// TIA Portal V15.1 export
// export: Created 2024-05-17T05:38:24.0424637Z, ExportSetting WithDefaults, DisplayName Totally Integrated Automation Portal, DisplayVersion V15.1 Update 5, DisplayName TIA Portal Openness, DisplayVersion V15.1 Update 5, DisplayName SINAMICS Startdrive Advanced, DisplayVersion V15.1, DisplayName G130, G150, S120, S150, SINAMICS MV, S210, DisplayVersion V15.1, DisplayName G110M, G120, G120C, G120D, G120P, DisplayVersion V15.1, DisplayName STEP 7 Professional, DisplayVersion V15.1 Update 5, DisplayName STEP 7 Safety, DisplayVersion V15.1, DisplayName WinCC Professional, DisplayVersion V15.1 Update 5, DisplayName SIMATIC Visualization Architect, DisplayVersion V15.1
FUNCTION "F209220ZS01Output" : Void   // FC7022, F_FBD
TITLE = Safety Inputs ZMProc / Safety Outputs 209220ZS01
{ S7_Optimized_Access := 'TRUE' }
VERSION : 0.1
// stored: AutoNumber false, IsIECCheckEnabled false, UDAEnableTagReadback false
BEGIN

REGION Network 1: **** --------------------- Infeed Roller // 220CR21 --------------------- ****
END_REGION

REGION Network 2: **** 8 - Outputs **** 209000AK04M1-UE140 Power OFF - 220CR21M1
   // SEW Drive Power OFF
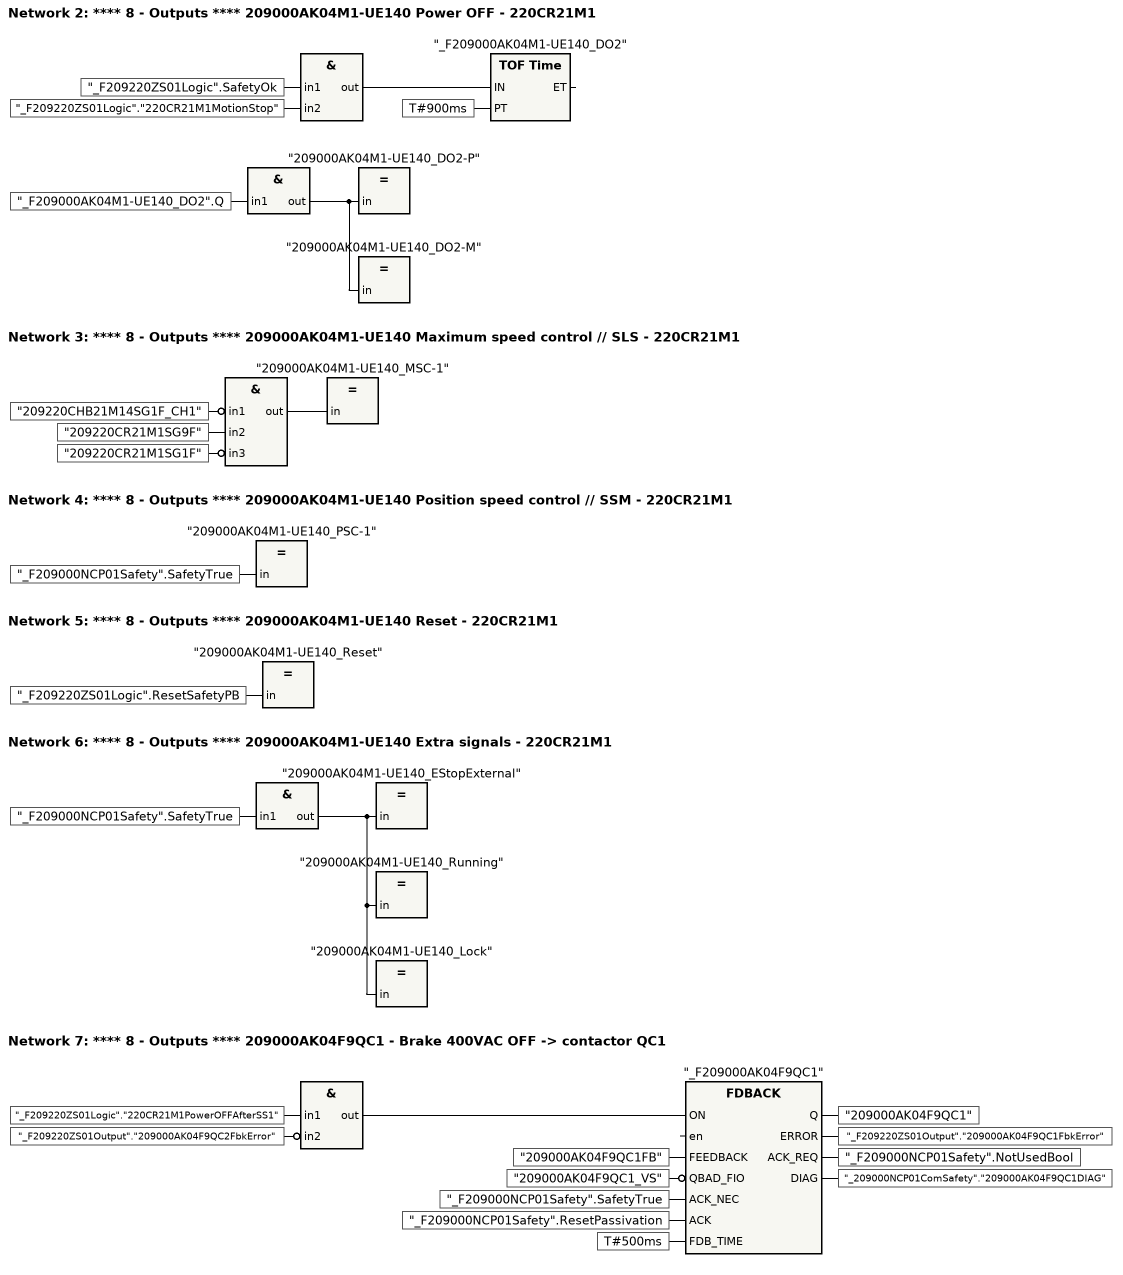
   "_F209000AK04M1-UE140_DO2".TOF(IN := "_F209220ZS01Logic".SafetyOk AND "_F209220ZS01Logic"."220CR21M1MotionStop",
                           PT := T#900ms);
   "209000AK04M1-UE140_DO2-P" := "_F209000AK04M1-UE140_DO2".Q;
   "209000AK04M1-UE140_DO2-M" := "_F209000AK04M1-UE140_DO2".Q;
END_REGION

REGION Network 3: **** 8 - Outputs **** 209000AK04M1-UE140 Maximum speed control // SLS - 220CR21M1
   // SEW Drive Maximum speed control
   "209000AK04M1-UE140_MSC-1" := NOT "209220CHB21M14SG1F_CH1" AND "209220CR21M1SG9F" AND NOT "209220CR21M1SG1F";
END_REGION

REGION Network 4: **** 8 - Outputs **** 209000AK04M1-UE140 Position speed control // SSM - 220CR21M1
   "209000AK04M1-UE140_PSC-1" := "_F209000NCP01Safety".SafetyTrue;
END_REGION

REGION Network 5: **** 8 - Outputs **** 209000AK04M1-UE140 Reset - 220CR21M1
   // SEW Drive Reset
   "209000AK04M1-UE140_Reset" := "_F209220ZS01Logic".ResetSafetyPB;
END_REGION

REGION Network 6: **** 8 - Outputs **** 209000AK04M1-UE140 Extra signals - 220CR21M1
   // SEW Drive Extra signals
   "209000AK04M1-UE140_EStopExternal" := "_F209000NCP01Safety".SafetyTrue;
   "209000AK04M1-UE140_Running" := "_F209000NCP01Safety".SafetyTrue;
   "209000AK04M1-UE140_Lock" := "_F209000NCP01Safety".SafetyTrue;
END_REGION

REGION Network 7: **** 8 - Outputs **** 209000AK04F9QC1 - Brake 400VAC OFF -> contactor QC1
   // Brake 400VAC OFF
   "_F209000AK04F9QC1"(ON := "_F209220ZS01Logic"."220CR21M1PowerOFFAfterSS1" AND NOT "_F209220ZS01Output"."209000AK04F9QC2FbkError",   // FDBACK
                       FEEDBACK := "209000AK04F9QC1FB",
                       QBAD_FIO := NOT "209000AK04F9QC1_VS",
                       ACK_NEC := "_F209000NCP01Safety".SafetyTrue,
                       ACK := "_F209000NCP01Safety".ResetPassivation,
                       FDB_TIME := T#500ms,
                       Q => "209000AK04F9QC1",
                       ERROR => "_F209220ZS01Output"."209000AK04F9QC1FbkError",
                       ACK_REQ => "_F209000NCP01Safety".NotUsedBool,
                       DIAG => "_209000NCP01ComSafety"."209000AK04F9QC1DIAG");
END_REGION

REGION Network 8: **** 8 - Outputs **** 209000AK04F9QC2 - Brake 400VAC OFF -> contactor QC2
   // Brake 400VAC OFF
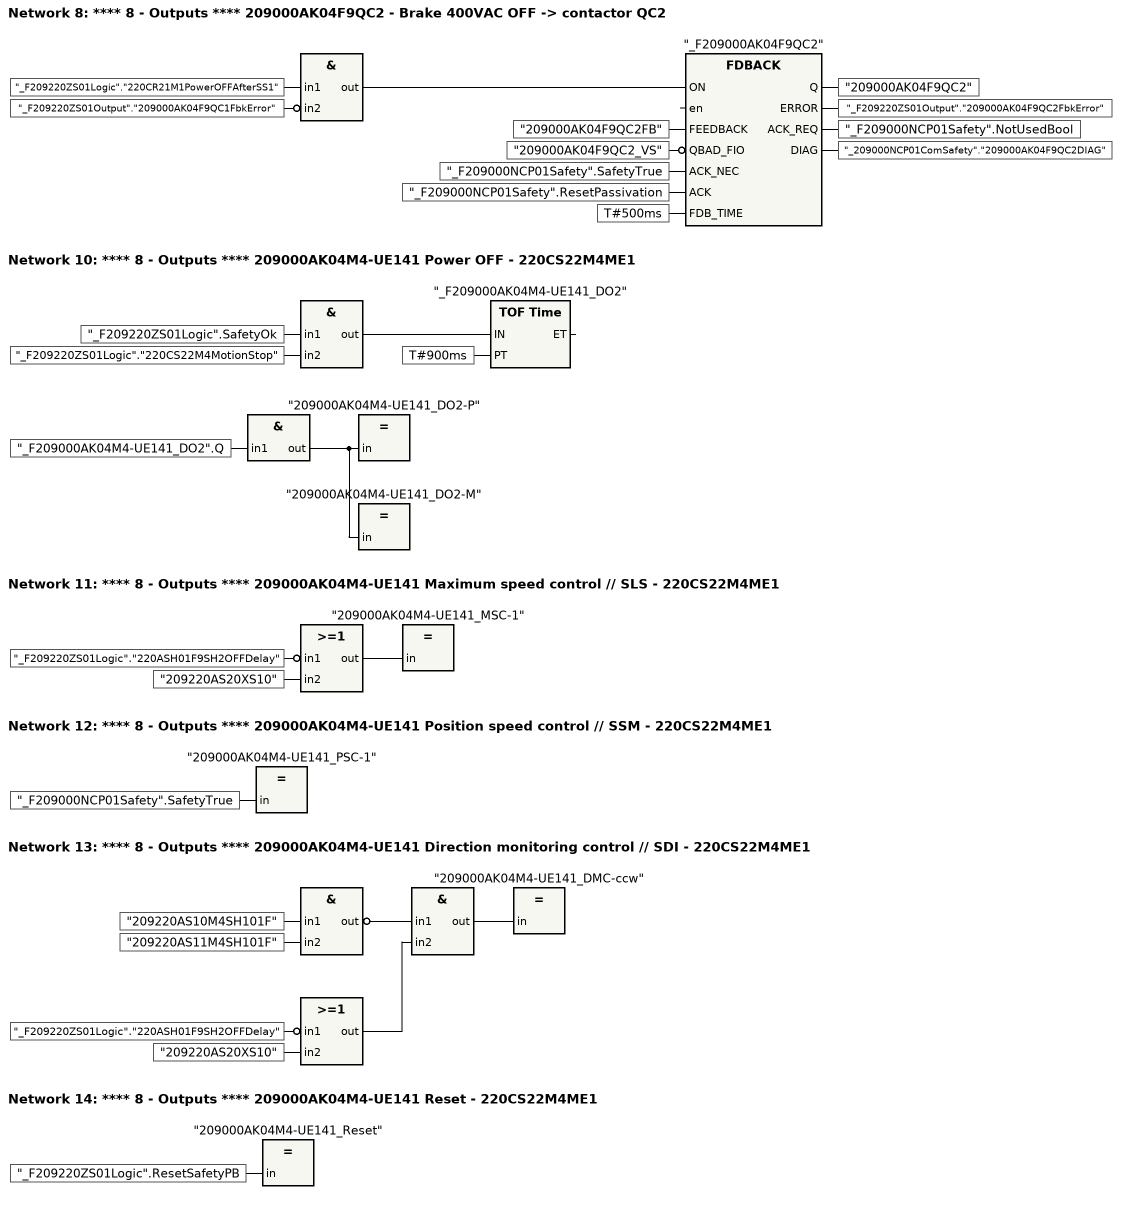
   "_F209000AK04F9QC2"(ON := "_F209220ZS01Logic"."220CR21M1PowerOFFAfterSS1" AND NOT "_F209220ZS01Output"."209000AK04F9QC1FbkError",   // FDBACK
                       FEEDBACK := "209000AK04F9QC2FB",
                       QBAD_FIO := NOT "209000AK04F9QC2_VS",
                       ACK_NEC := "_F209000NCP01Safety".SafetyTrue,
                       ACK := "_F209000NCP01Safety".ResetPassivation,
                       FDB_TIME := T#500ms,
                       Q => "209000AK04F9QC2",
                       ERROR => "_F209220ZS01Output"."209000AK04F9QC2FbkError",
                       ACK_REQ => "_F209000NCP01Safety".NotUsedBool,
                       DIAG => "_209000NCP01ComSafety"."209000AK04F9QC2DIAG");
END_REGION

REGION Network 9: **** --------------------- Slat Conveyor // 220CS22 --------------------- ****
END_REGION

REGION Network 10: **** 8 - Outputs **** 209000AK04M4-UE141 Power OFF - 220CS22M4ME1
   // SEW Drive Power OFF
   "_F209000AK04M4-UE141_DO2".TOF(IN := "_F209220ZS01Logic".SafetyOk AND "_F209220ZS01Logic"."220CS22M4MotionStop",
                           PT := T#900ms);
   "209000AK04M4-UE141_DO2-P" := "_F209000AK04M4-UE141_DO2".Q;
   "209000AK04M4-UE141_DO2-M" := "_F209000AK04M4-UE141_DO2".Q;
END_REGION

REGION Network 11: **** 8 - Outputs **** 209000AK04M4-UE141 Maximum speed control // SLS - 220CS22M4ME1
   // SEW Drive Maximum speed control
   "209000AK04M4-UE141_MSC-1" := NOT "_F209220ZS01Logic"."220ASH01F9SH2OFFDelay" OR "209220AS20XS10";
END_REGION

REGION Network 12: **** 8 - Outputs **** 209000AK04M4-UE141 Position speed control // SSM - 220CS22M4ME1
   "209000AK04M4-UE141_PSC-1" := "_F209000NCP01Safety".SafetyTrue;
END_REGION

REGION Network 13: **** 8 - Outputs **** 209000AK04M4-UE141 Direction monitoring control // SDI - 220CS22M4ME1
   "209000AK04M4-UE141_DMC-ccw" := NOT ("209220AS10M4SH101F" AND "209220AS11M4SH101F") AND (NOT "_F209220ZS01Logic"."220ASH01F9SH2OFFDelay" OR "209220AS20XS10");
END_REGION

REGION Network 14: **** 8 - Outputs **** 209000AK04M4-UE141 Reset - 220CS22M4ME1
   // SEW Drive Reset
   "209000AK04M4-UE141_Reset" := "_F209220ZS01Logic".ResetSafetyPB;
END_REGION

REGION Network 15: **** 8 - Outputs **** 209000AK04M4-UE141 Extra signals - 220CS22M4ME1
   // SEW Drive Extra signals
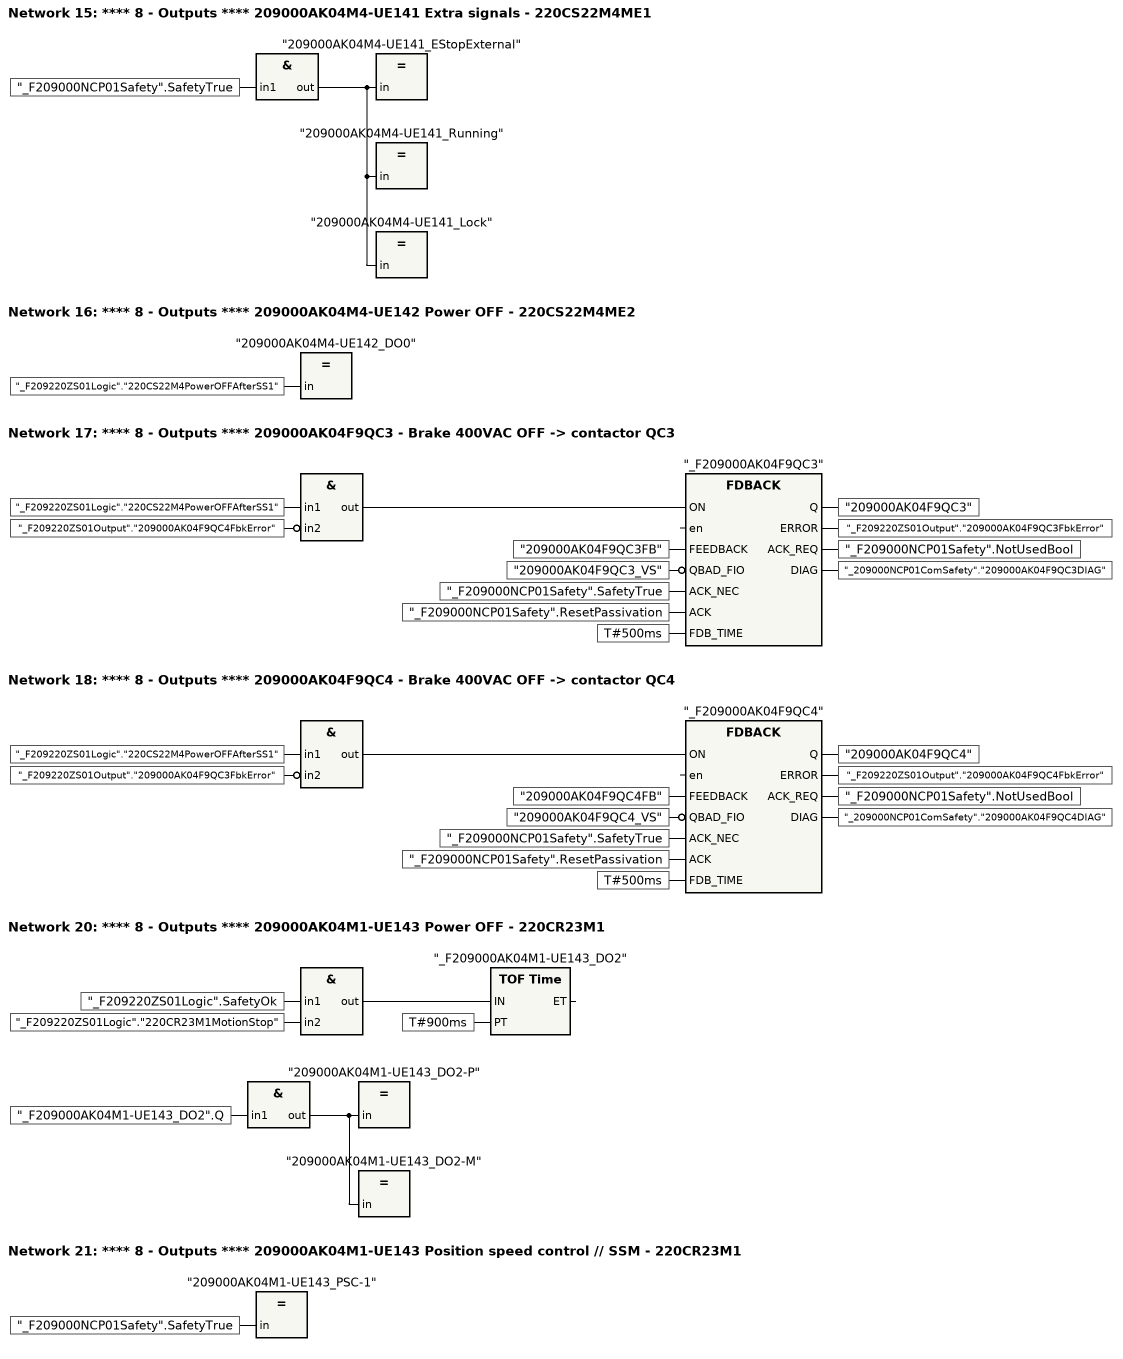
   "209000AK04M4-UE141_EStopExternal" := "_F209000NCP01Safety".SafetyTrue;
   "209000AK04M4-UE141_Running" := "_F209000NCP01Safety".SafetyTrue;
   "209000AK04M4-UE141_Lock" := "_F209000NCP01Safety".SafetyTrue;
END_REGION

REGION Network 16: **** 8 - Outputs **** 209000AK04M4-UE142 Power OFF - 220CS22M4ME2
   // SEW Drive Power OFF
   "209000AK04M4-UE142_DO0" := "_F209220ZS01Logic"."220CS22M4PowerOFFAfterSS1";
END_REGION

REGION Network 17: **** 8 - Outputs **** 209000AK04F9QC3 - Brake 400VAC OFF -> contactor QC3
   // Brake 400VAC OFF
   "_F209000AK04F9QC3"(ON := "_F209220ZS01Logic"."220CS22M4PowerOFFAfterSS1" AND NOT "_F209220ZS01Output"."209000AK04F9QC4FbkError",   // FDBACK
                       FEEDBACK := "209000AK04F9QC3FB",
                       QBAD_FIO := NOT "209000AK04F9QC3_VS",
                       ACK_NEC := "_F209000NCP01Safety".SafetyTrue,
                       ACK := "_F209000NCP01Safety".ResetPassivation,
                       FDB_TIME := T#500ms,
                       Q => "209000AK04F9QC3",
                       ERROR => "_F209220ZS01Output"."209000AK04F9QC3FbkError",
                       ACK_REQ => "_F209000NCP01Safety".NotUsedBool,
                       DIAG => "_209000NCP01ComSafety"."209000AK04F9QC3DIAG");
END_REGION

REGION Network 18: **** 8 - Outputs **** 209000AK04F9QC4 - Brake 400VAC OFF -> contactor QC4
   // Brake 400VAC OFF
   "_F209000AK04F9QC4"(ON := "_F209220ZS01Logic"."220CS22M4PowerOFFAfterSS1" AND NOT "_F209220ZS01Output"."209000AK04F9QC3FbkError",   // FDBACK
                       FEEDBACK := "209000AK04F9QC4FB",
                       QBAD_FIO := NOT "209000AK04F9QC4_VS",
                       ACK_NEC := "_F209000NCP01Safety".SafetyTrue,
                       ACK := "_F209000NCP01Safety".ResetPassivation,
                       FDB_TIME := T#500ms,
                       Q => "209000AK04F9QC4",
                       ERROR => "_F209220ZS01Output"."209000AK04F9QC4FbkError",
                       ACK_REQ => "_F209000NCP01Safety".NotUsedBool,
                       DIAG => "_209000NCP01ComSafety"."209000AK04F9QC4DIAG");
END_REGION

REGION Network 19: **** --------------------- Outfeed Roller // 220CR23 --------------------- ****
END_REGION

REGION Network 20: **** 8 - Outputs **** 209000AK04M1-UE143 Power OFF - 220CR23M1
   // SEW Drive Power OFF
   "_F209000AK04M1-UE143_DO2".TOF(IN := "_F209220ZS01Logic".SafetyOk AND "_F209220ZS01Logic"."220CR23M1MotionStop",
                           PT := T#900ms);
   "209000AK04M1-UE143_DO2-P" := "_F209000AK04M1-UE143_DO2".Q;
   "209000AK04M1-UE143_DO2-M" := "_F209000AK04M1-UE143_DO2".Q;
END_REGION

REGION Network 21: **** 8 - Outputs **** 209000AK04M1-UE143 Position speed control // SSM - 220CR23M1
   "209000AK04M1-UE143_PSC-1" := "_F209000NCP01Safety".SafetyTrue;
END_REGION

REGION Network 22: **** 8 - Outputs **** 209000AK04M1-UE143 Direction monitoring control // SDI - 220CR23M1
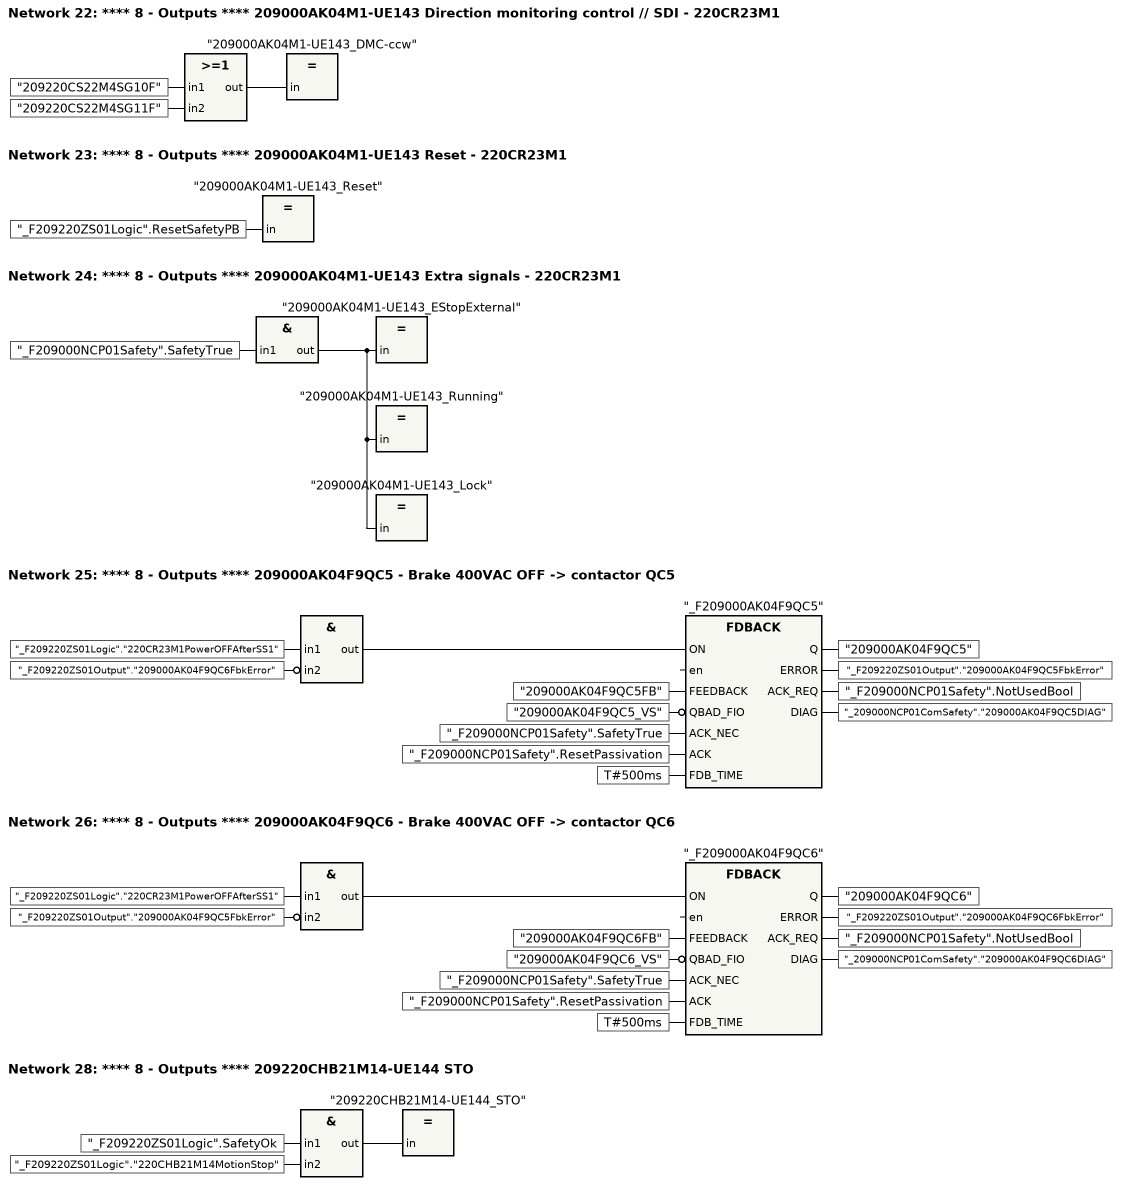
   "209000AK04M1-UE143_DMC-ccw" := "209220CS22M4SG10F" OR "209220CS22M4SG11F";
END_REGION

REGION Network 23: **** 8 - Outputs **** 209000AK04M1-UE143 Reset - 220CR23M1
   // SEW Drive Reset
   "209000AK04M1-UE143_Reset" := "_F209220ZS01Logic".ResetSafetyPB;
END_REGION

REGION Network 24: **** 8 - Outputs **** 209000AK04M1-UE143 Extra signals - 220CR23M1
   // SEW Drive Extra signals
   "209000AK04M1-UE143_EStopExternal" := "_F209000NCP01Safety".SafetyTrue;
   "209000AK04M1-UE143_Running" := "_F209000NCP01Safety".SafetyTrue;
   "209000AK04M1-UE143_Lock" := "_F209000NCP01Safety".SafetyTrue;
END_REGION

REGION Network 25: **** 8 - Outputs **** 209000AK04F9QC5 - Brake 400VAC OFF -> contactor QC5
   // Brake 400VAC OFF
   "_F209000AK04F9QC5"(ON := "_F209220ZS01Logic"."220CR23M1PowerOFFAfterSS1" AND NOT "_F209220ZS01Output"."209000AK04F9QC6FbkError",   // FDBACK
                       FEEDBACK := "209000AK04F9QC5FB",
                       QBAD_FIO := NOT "209000AK04F9QC5_VS",
                       ACK_NEC := "_F209000NCP01Safety".SafetyTrue,
                       ACK := "_F209000NCP01Safety".ResetPassivation,
                       FDB_TIME := T#500ms,
                       Q => "209000AK04F9QC5",
                       ERROR => "_F209220ZS01Output"."209000AK04F9QC5FbkError",
                       ACK_REQ => "_F209000NCP01Safety".NotUsedBool,
                       DIAG => "_209000NCP01ComSafety"."209000AK04F9QC5DIAG");
END_REGION

REGION Network 26: **** 8 - Outputs **** 209000AK04F9QC6 - Brake 400VAC OFF -> contactor QC6
   // Brake 400VAC OFF
   "_F209000AK04F9QC6"(ON := "_F209220ZS01Logic"."220CR23M1PowerOFFAfterSS1" AND NOT "_F209220ZS01Output"."209000AK04F9QC5FbkError",   // FDBACK
                       FEEDBACK := "209000AK04F9QC6FB",
                       QBAD_FIO := NOT "209000AK04F9QC6_VS",
                       ACK_NEC := "_F209000NCP01Safety".SafetyTrue,
                       ACK := "_F209000NCP01Safety".ResetPassivation,
                       FDB_TIME := T#500ms,
                       Q => "209000AK04F9QC6",
                       ERROR => "_F209220ZS01Output"."209000AK04F9QC6FbkError",
                       ACK_REQ => "_F209000NCP01Safety".NotUsedBool,
                       DIAG => "_209000NCP01ComSafety"."209000AK04F9QC6DIAG");
END_REGION

REGION Network 27: **** --------------------- Hold Back // 220CHB21 --------------------- ****
END_REGION

REGION Network 28: **** 8 - Outputs **** 209220CHB21M14-UE144 STO
   // SEW Drive STO
   "209220CHB21M14-UE144_STO" := "_F209220ZS01Logic".SafetyOk AND "_F209220ZS01Logic"."220CHB21M14MotionStop";
END_REGION
END_FUNCTION
